// TIA Portal project "ZápisDB" (V14)

(* hardware
DEVICE "ET 200S station_1"  ET 200S station
   slot 0: "Rack_0"  Rail
   slot 2: "PLC_1"  IM 151-8 PN/DP CPU  6ES7 151-8AB01-0AB0  V3.2
      slot 1: "PROFINET interface_1"  PN-IO
         slot 1: "Port_1"  Port
         slot 2: "Port_2"  Port
         slot 3: "Port_3"  Port
DEVICE "S71500/ET200MP station_1"  S7-1500 station
   slot 0: "Rail_0"  Rack  6ES7 590-1***0-0AA0
   slot 1: "PLC_2"  CPU 1511-1 PN  6ES7 511-1AK01-0AB0  V2.1
      slot 3: "CPU display_1"  6ES7591-1AA00-0AA0
DEVICE "S7300/ET200M station_1"  S7-300 station
   slot 0: "Rail_0"  Rail  6ES7 390-1***0-0AA0
   slot 2: "PLC_3"  CPU 312  6ES7 312-1AE14-0AB0  V3.3
      slot 0: "MPI interface_1"  MPI
DEVICE "S7-1200 station_1"  S7-1200 Station
   slot 0: "Rack_0"  S7-1200 Rack  Rack  V1.0
   slot 1: "PLC_4"  CPU 1211C AC/DC/Rly  6ES7 211-1BE40-0XB0  V4.2
*)

// ===== PLC "PLC_1"  IM 151-8 PN/DP CPU =====

VAR_GLOBAL   // PLC tag table "Default tag table"
   "Tag_1" AT %M10.0 : Bool;
   "Tag_2" AT %M10.1 : Bool;
   "Tag_3" AT %MB200 : Byte;
   "Tag_4" AT %M0.0 : Bool;
   "Tag_5" AT %M1.0 : Bool;
   "Tag_6" AT %M1.2 : Bool;
END_VAR

TYPE "Objekt"
   STRUCT
      Velikost : Int;
      Pocet : Int;
   END_STRUCT;
END_TYPE

TYPE "User_data_type_1"
   STRUCT
      aa : Bool;
   END_STRUCT;
END_TYPE

DATA_BLOCK "CreateDB_DB"   // DB1
{ S7_Optimized_Access := 'FALSE' }
VERSION : 0.1
// stored: InstanceOfName CreateDB
"CreateDB"
BEGIN
END_DATA_BLOCK

DATA_BLOCK "Block_1_DB"   // DB2
{ S7_Optimized_Access := 'FALSE' }
VERSION : 0.1
// stored: InstanceOfName Block_1
"Block_1"
BEGIN
END_DATA_BLOCK

DATA_BLOCK "Block_1_DB_1"   // DB3
{ S7_Optimized_Access := 'FALSE' }
VERSION : 0.1
// stored: InstanceOfName Block_1
"Block_1"
BEGIN
END_DATA_BLOCK

DATA_BLOCK "Data_block_3"   // DB4
{ S7_Optimized_Access := 'FALSE' }
VERSION : 0.1
   VAR
      aa : Bool;
   END_VAR
BEGIN
END_DATA_BLOCK

DATA_BLOCK "Data_block_4"   // DB5
{ S7_Optimized_Access := 'FALSE' }
VERSION : 0.1
BEGIN
END_DATA_BLOCK

DATA_BLOCK "Data_block_1"   // DB10
{ S7_Optimized_Access := 'FALSE' }
VERSION : 0.1
   VAR
      aa : Word;
      dd : Word;
      ee : Word;
      kk : Word;
   END_VAR
BEGIN
END_DATA_BLOCK

DATA_BLOCK "Data_block_2"   // DB11
{ S7_Optimized_Access := 'FALSE' }
VERSION : 0.1
   VAR
      aa : Word;
      dd : Word;
      ee : Word;
      ll : Word;
   END_VAR
BEGIN
END_DATA_BLOCK

DATA_BLOCK "Source"   // DB100
{ S7_Optimized_Access := 'FALSE' }
VERSION : 0.1
   VAR
      Object : "Objekt";
   END_VAR
BEGIN
END_DATA_BLOCK

DATA_BLOCK "Data"   // DB101
{ S7_Optimized_Access := 'FALSE' }
VERSION : 0.1
   VAR
      eeee : Bool;
   END_VAR
BEGIN
END_DATA_BLOCK

FUNCTION_BLOCK "CreateDB"   // FB1, LAD
{ S7_Optimized_Access := 'FALSE' }
VERSION : 0.1
   VAR_INPUT
      object : "Objekt";
   END_VAR
   VAR_TEMP
      number : Word;
      aa : Bool;
      error : Int;
      busy : Bool;
   END_VAR
   VAR_TEMP   // added for the SCL form of the ladder/FBD networks
      _w1 : Bool;
   END_VAR
BEGIN

REGION Network 1
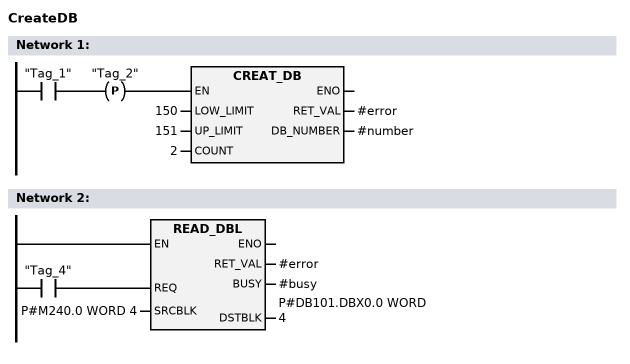
   #_w1 := "Tag_1" AND NOT "Tag_2";   // rising edge
   "Tag_2" := "Tag_1";
   IF #_w1 THEN
       #error := CREAT_DB(LOW_LIMIT := 150, UP_LIMIT := 151, COUNT := 2, DB_NUMBER => #number);
   END_IF;
END_REGION

REGION Network 2
   #error := READ_DBL(REQ := "Tag_4", SRCBLK := P#M240.0 WORD 4, BUSY => #busy, DSTBLK => P#DB101.DBX0.0 WORD 4);
END_REGION
END_FUNCTION_BLOCK

FUNCTION_BLOCK "Block_1"   // FB2, STL
{ S7_Optimized_Access := 'FALSE' }
VERSION : 0.1
   VAR_INPUT
      Input_1 : Block_SDB;
      aa : Int;
   END_VAR
   VAR_TEMP
      "lokální 1" : Int;
      další : Int;
   END_VAR
BEGIN

REGION Network 1
         L     99;
         T     #"lokální 1";


         L     #"lokální 1";
         T     "Tag_3";
END_REGION
END_FUNCTION_BLOCK

FUNCTION_BLOCK "Enot"   // FB3, LAD
{ S7_Optimized_Access := 'FALSE' }
VERSION : 0.1
BEGIN

REGION Network 1
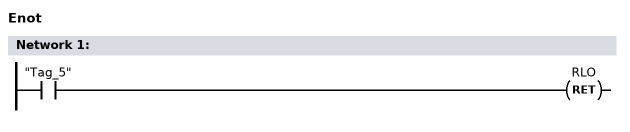
   IF "Tag_5" THEN
       ENO := TRUE;
       RETURN;
   END_IF;
END_REGION
END_FUNCTION_BLOCK

FUNCTION_BLOCK "Block_2"   // FB4, FBD
{ S7_Optimized_Access := 'FALSE' }
VERSION : 0.1
BEGIN
END_FUNCTION_BLOCK

ORGANIZATION_BLOCK "Main"   // OB1, LAD
TITLE = "Main Program Sweep (Cycle)"
{ S7_Optimized_Access := 'FALSE' }
VERSION : 0.1
   VAR_TEMP
      OB1_EV_CLASS : Byte;   // Bits 0-3 = 1 (Coming event), Bits 4-7 = 1 (Event class 1)
      OB1_SCAN_1 : Byte;   // 1 (Cold restart scan 1 of OB 1), 3 (Scan 2-n of OB 1)
      OB1_PRIORITY : Byte;   // Priority of OB Execution
      OB1_OB_NUMBR : Byte;   // 1 (Organization block 1, OB1)
      OB1_RESERVED_1 : Byte;   // Reserved for system
      OB1_RESERVED_2 : Byte;   // Reserved for system
      OB1_PREV_CYCLE : Int;   // Cycle time of previous OB1 scan (milliseconds)
      OB1_MIN_CYCLE : Int;   // Minimum cycle time of OB1 (milliseconds)
      OB1_MAX_CYCLE : Int;   // Maximum cycle time of OB1 (milliseconds)
      OB1_DATE_TIME : Date_And_Time;   // Date and time OB1 started
   END_VAR
BEGIN

REGION Network 1
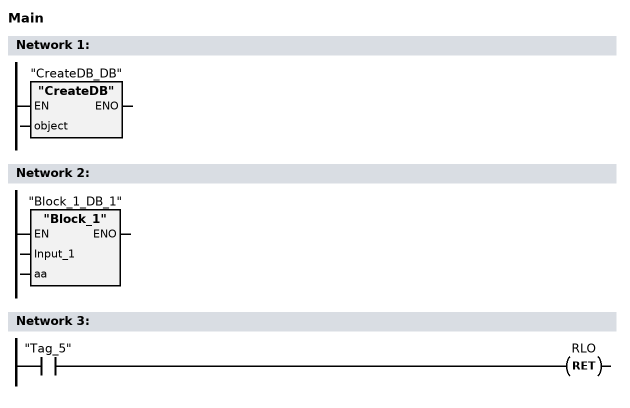
   RUNG wire#powerrail
      "CreateDB_DB"(object :=)
   END_RUNG
   // the same network as SCL:
   "CreateDB_DB"();   // "CreateDB"
END_REGION

REGION Network 2
   RUNG wire#powerrail
      "Block_1_DB_1"(Input_1 :=, aa :=)
   END_RUNG
   // the same network as SCL:
   "Block_1_DB_1"();   // "Block_1"
END_REGION

REGION Network 3
   IF "Tag_5" THEN
       ENO := TRUE;
       RETURN;
   END_IF;
END_REGION
END_ORGANIZATION_BLOCK

// ===== PLC "PLC_2"  CPU 1511-1 PN =====

VAR_GLOBAL   // PLC tag table "Default tag table"
   "Tag_1" AT %M1.0 : Bool;
   "Tag_2" AT %M90.0 : Bool;
END_VAR

TYPE "User_data_type_1"
   STRUCT
      aaaa : Bool;
   END_STRUCT;
END_TYPE

TYPE "User_data_type_2"
   STRUCT
      Element_1 : Event_Any;
   END_STRUCT;
END_TYPE

TYPE "User_data_type_3"
END_TYPE

DATA_BLOCK "Block_2_DB"   // DB2
{ S7_Optimized_Access := 'TRUE' }
VERSION : 0.1
// stored: InstanceOfName Block_2
"Block_2"
BEGIN
END_DATA_BLOCK

DATA_BLOCK "Block_5_DB"   // DB3
{ S7_Optimized_Access := 'TRUE' }
VERSION : 0.1
// stored: InstanceOfName Block_5
"Block_5"
BEGIN
END_DATA_BLOCK

DATA_BLOCK "Data_block_1"   // DB4
{ S7_Optimized_Access := 'TRUE' }
VERSION : 0.1
BEGIN
END_DATA_BLOCK

FUNCTION_BLOCK "Block_1"   // FB1, LAD
{ S7_Optimized_Access := 'TRUE' }
VERSION : 0.1
BEGIN

REGION Network 1
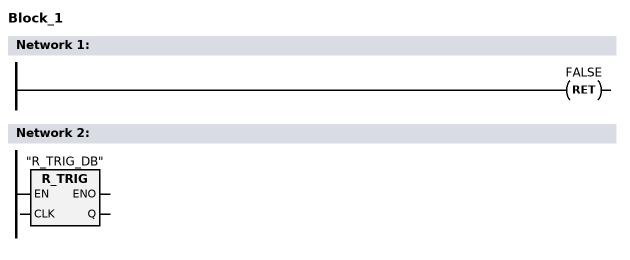
   ENO := FALSE;
   RETURN;
END_REGION

REGION Network 2
   "R_TRIG_DB"();   // R_TRIG
END_REGION
END_FUNCTION_BLOCK

FUNCTION_BLOCK "Block_2"   // FB2, ProDiag
{ S7_Optimized_Access := 'TRUE' }
VERSION : 0.1
   VAR
      State : SV_FB_State;
      Tag_1_O_1 : SV_State;
   END_VAR
   VAR_TEMP
      t_TempSvStateUDT : SV_State;
      t_TempAlarmInstance : <type 200004f>;
      t_TempAsocValue1 : Variant;
      t_TempAsocValue2 : Variant;
      t_TempAsocValue3 : Variant;
   END_VAR
BEGIN
END_FUNCTION_BLOCK

FUNCTION_BLOCK "Block_3"   // FB3, SCL
{ S7_Optimized_Access := 'TRUE' }
VERSION : 0.1
BEGIN
END_FUNCTION_BLOCK

FUNCTION_BLOCK "Block_4"   // FB4, LAD
{ S7_Optimized_Access := 'TRUE' }
VERSION : 0.1
BEGIN
END_FUNCTION_BLOCK

FUNCTION_BLOCK "Block_5"   // FB5, ProDiag
{ S7_Optimized_Access := 'TRUE' }
VERSION : 0.1
   VAR
      State : SV_FB_State;
      Tag_2_A_1 : SV_State;
      Tag_2_O_1 : SV_State;
   END_VAR
   VAR_TEMP
      t_TempSvStateUDT : SV_State;
      t_TempAlarmInstance : <type 200004f>;
      t_TempAsocValue1 : Variant;
      t_TempAsocValue2 : Variant;
      t_TempAsocValue3 : Variant;
   END_VAR
BEGIN
END_FUNCTION_BLOCK

FUNCTION_BLOCK "Block_6"   // FB6, LAD
{ S7_Optimized_Access := 'TRUE' }
VERSION : 0.1
   VAR_IN_OUT
      io : Bool;
   END_VAR
BEGIN
END_FUNCTION_BLOCK

ORGANIZATION_BLOCK "Main"   // OB1, LAD, ProgramCycle
TITLE = "Main Program Sweep (Cycle)"
{ S7_Optimized_Access := 'TRUE' }
VERSION : 0.1
   VAR_INPUT
      Initial_Call : Bool;   // Initial call of this OB
      Remanence : Bool;   // =True, if remanent data are available
   END_VAR
BEGIN
END_ORGANIZATION_BLOCK

// ===== PLC "PLC_3"  CPU 312 =====

ORGANIZATION_BLOCK "Main"   // OB1, LAD
TITLE = "Main Program Sweep (Cycle)"
{ S7_Optimized_Access := 'FALSE' }
VERSION : 0.1
   VAR_TEMP
      OB1_EV_CLASS : Byte;   // Bits 0-3 = 1 (Coming event), Bits 4-7 = 1 (Event class 1)
      OB1_SCAN_1 : Byte;   // 1 (Cold restart scan 1 of OB 1), 3 (Scan 2-n of OB 1)
      OB1_PRIORITY : Byte;   // Priority of OB Execution
      OB1_OB_NUMBR : Byte;   // 1 (Organization block 1, OB1)
      OB1_RESERVED_1 : Byte;   // Reserved for system
      OB1_RESERVED_2 : Byte;   // Reserved for system
      OB1_PREV_CYCLE : Int;   // Cycle time of previous OB1 scan (milliseconds)
      OB1_MIN_CYCLE : Int;   // Minimum cycle time of OB1 (milliseconds)
      OB1_MAX_CYCLE : Int;   // Maximum cycle time of OB1 (milliseconds)
      OB1_DATE_TIME : Date_And_Time;   // Date and time OB1 started
   END_VAR
BEGIN
END_ORGANIZATION_BLOCK

// ===== PLC "PLC_4"  CPU 1211C AC/DC/Rly =====

VAR_GLOBAL   // PLC tag table "Default tag table"
   "Tag_1" AT %M1.0 : Bool;
END_VAR

FUNCTION_BLOCK "Block_1"   // FB1, LAD
{ S7_Optimized_Access := 'TRUE' }
VERSION : 0.1
BEGIN

REGION Network 1
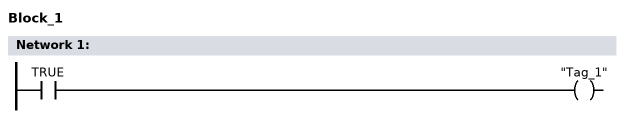
   RUNG wire#powerrail
      Contact( TRUE )
      Coil( "Tag_1" )
   END_RUNG
   // the same network as SCL:
   "Tag_1" := TRUE;
END_REGION
END_FUNCTION_BLOCK

FUNCTION_BLOCK "Block_2"   // FB2, LAD
{ S7_Optimized_Access := 'TRUE' }
VERSION : 0.1
BEGIN
END_FUNCTION_BLOCK

ORGANIZATION_BLOCK "Main"   // OB1, LAD, ProgramCycle
TITLE = "Main Program Sweep (Cycle)"
{ S7_Optimized_Access := 'TRUE' }
VERSION : 0.1
   VAR_INPUT
      Initial_Call : Bool;   // Initial call of this OB
      Remanence : Bool;   // =True, if remanent data are available
   END_VAR
BEGIN
END_ORGANIZATION_BLOCK